PROGRAM PROP_BARCODE_MAIN
VAR
	barcodeState : E_Barcode_State := E_Barcode_State.INIT;
	
	newData_Front : BYTE := 16#00;
	newData_Back : BYTE := 16#00;
	
	positionValues_Front : ARRAY[0..3] OF BYTE;
	velocityValues_Front : ARRAY[0..1] OF BYTE; 
	
	positionValues_Back : ARRAY[0..3] OF BYTE;
	velocityValues_Back : ARRAY[0..1] OF BYTE; 
	
	position_Front : DINT;
	position_Back : DINT;
	
	velocity_Front : DINT;
	velocity_BacK : DINT;
	
	start : BOOL := FALSE;
END_VAR
VAR CONSTANT
	SCALE_FACTOR : INT := 100;
	BARCODE_START : INT := 11920;
	SET_COMMAND : BYTE := 16#01;
	SEND_POS_VEL : BYTE := 16#80;
	SEND_DIAG : BYTE := 16#08;
	SEND_MARKER_INFO : BYTE := 16#02;
END_VAR

CASE barcodeState OF
	
	E_Barcode_State.INIT:
	
		IF start THEN
			barcodeState := E_BARCODE_STATE.SEND_POS_VEL_COMMAND;
		END_IF
		
	E_Barcode_State.SEND_POS_VEL_COMMAND:
		
		positionValues_Front[0] := GVL_PROP.InputData1_Front[4];
		positionValues_Front[1] := GVL_PROP.InputData1_Front[5];
		positionValues_Front[2] := GVL_PROP.InputData1_Front[6];
		positionValues_Front[3] := GVL_PROP.InputData1_Front[7];
		
		velocityValues_Front[0] := GVL_PROP.InputData2_Front[0];
		velocityValues_Front[1] := GVL_PROP.InputData2_Front[1];
		
//-----------------------
		
		positionValues_Back[0] := GVL_PROP.InputData1_Front[4];
		positionValues_Back[1] := GVL_PROP.InputData1_Front[5];
		positionValues_Back[2] := GVL_PROP.InputData1_Front[6];
		positionValues_Back[3] := GVL_PROP.InputData1_Front[7];
		
		velocityValues_Back[0] := GVL_PROP.InputData2_Front[0];
		velocityValues_Back[1] := GVL_PROP.InputData2_Front[1];
		
//-----------------------		

		IF velocityValues_Front[0] > 128 THEN
			velocity_Front := (256 * 256 - (256 * velocityValues_Front[0] + velocityValues_Front[1]));
		ELSE
			velocity_Front := 256 * velocityValues_Front[0] + velocityValues_Front[1];	
		END_IF
		
		position_Front := 
			256 * 256 * 256 * positionValues_Front[0]
			+ 256 * 256 * positionValues_Front[1]
			+ 256 * positionValues_Front[2]
			+ positionValues_Front[3];
			
		position_Front := position_Front / SCALE_FACTOR - BARCODE_START;
		
//------------------------		

		IF velocityValues_Back[0] > 128 THEN
			velocity_Back := (256 * 256 - (256 * velocityValues_Back[0] + velocityValues_Back[1]));
		ELSE
			velocity_Back := 256 * velocityValues_Back[0] + velocityValues_Back[1];	
		END_IF
		
		position_Back := 
			256 * 256 * 256 * positionValues_Back[0]
			+ 256 * 256 * positionValues_Back[1]
			+ 256 * positionValues_Back[2]
			+ positionValues_Back[3];
			
		position_Back := position_Back / SCALE_FACTOR - BARCODE_START;
		
		newData_Back := newData_Back XOR 16#80;
		
		GVL_PROP.OutputData_Back[0] := newData_Back OR SET_COMMAND;
		GVL_PROP.OutputData_Back[2] := SEND_POS_VEL;
		
//unsure what this is used for 		
	E_Barcode_State.SEND_DIAGNOSTIC_COMMAND:
	
		newData_Front := newData_Front XOR 16#80;
		
		GVL_PROP.OutputData_Front[0] := newData_Front OR SET_COMMAND;
		GVL_PROP.OutputData_Front[2] := 16#00;
		GVL_PROP.OutputData_Front[3] := SEND_DIAG;

//-------------------------
		
		newData_Back := newData_Back XOR 16#80;
		
		GVL_PROP.OutputData_Back[0] := newData_Back OR SET_COMMAND;
		GVL_PROP.OutputData_Back[2] := 16#00;
		GVL_PROP.OutputData_Back[3] := SEND_DIAG;

	
//unsure what this is used for 		
	E_Barcode_State.SEND_MARKER_INFO_COMMAND:
	
		newData_Front := newData_Front XOR 16#80;
		GVL_PROP.OutputData_Front[0] := newData_Front OR SET_COMMAND;
		GVL_PROP.OutputData_Front[2] := 16#00;
		GVL_PROP.OutputData_Front[3] := SEND_MARKER_INFO;
		
//------------------------
		
		newData_Back := newData_Back XOR 16#80;
		GVL_PROP.OutputData_Back[0] := newData_Front OR SET_COMMAND;
		GVL_PROP.OutputData_Back[2] := 16#00;
		GVL_PROP.OutputData_Back[3] := SEND_MARKER_INFO;

		
	E_Barcode_State.ERROR:
		barcodeState := E_Barcode_State.INIT;
		start := FALSE;
	
END_CASE

END_PROGRAM

(* stored: Version 1.1.0.1
   POU PROP_BARCODE_MAIN: Id {c5354a79-cedd-4abc-9f85-b60d39285641}, SpecialFunc None *)
